// Mitsubishi GX Works2 project: Test Module 64AD   PLC: Q03UDV
// 20181022A

PROGRAM 64AD
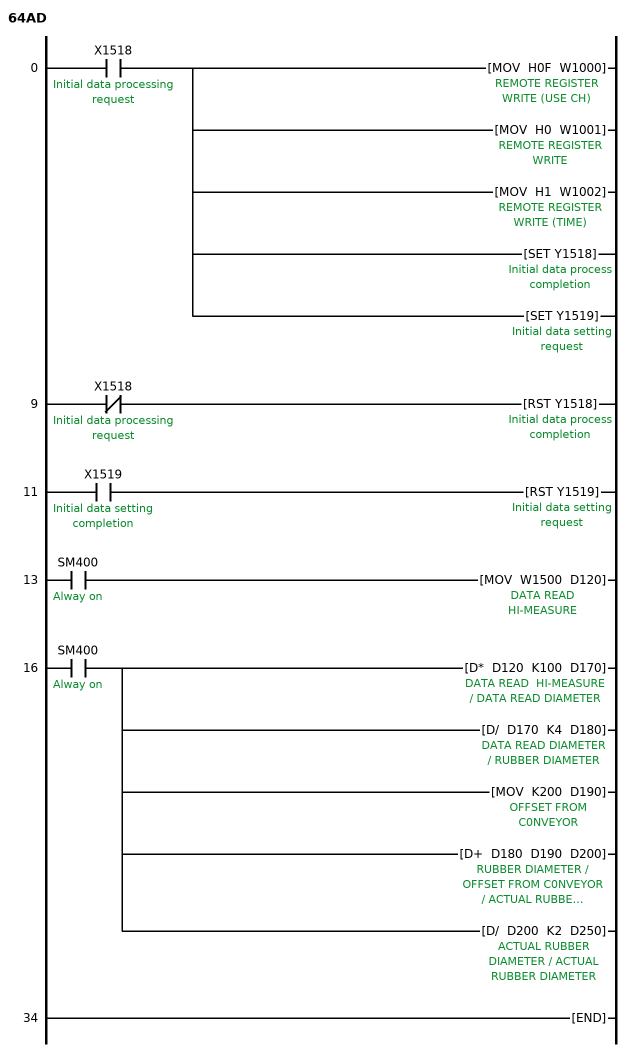
0     LD      X1518  ; Initial data processing request
      MOV     H0F W1000  ; REMOTE REGISTER WRITE (USE CH)
      MOV     H0 W1001  ; REMOTE REGISTER WRITE
      MOV     H1 W1002  ; REMOTE REGISTER WRITE (TIME)
      SET     Y1518  ; Initial data process completion
      SET     Y1519  ; Initial data setting request
9     LDI     X1518  ; Initial data processing request
      RST     Y1518  ; Initial data process completion
11    LD      X1519  ; Initial data setting completion
      RST     Y1519  ; Initial data setting request
13    LD      SM400  ; Alway on
      MOV     W1500 D120  ; DATA READ  HI-MEASURE
16    LD      SM400  ; Alway on
      D*      D120 K100 D170  ; DATA READ DIAMETER
      D/      D170 K4 D180  ; RUBBER DIAMETER
      MOV     K200 D190  ; OFFSET FROM C0NVEYOR
      D+      D180 D190 D200  ; ACTUAL RUBBER DIAMETER
      D/      D200 K2 D250  ; ACTUAL RUBBER DIAMETER
34    END
END_PROGRAM
